FUNCTION_BLOCK AX_ATM_FB_TON (* standard timer function block (on-delay timing) with AX/ATM Adapter, PT and ET as adapters *)
  (* Standard: 61131-3; Classification: standard timer function block; Description: Copyright (c) 2026 HR Agrartechnik GmbH This program and the accompanying materials are made available under the terms of the Eclipse Public License 2.0 which is available at https://www.eclipse.org/legal/epl-2.0/ SPDX-License-Identifier: EPL-2.0 Wie AX_FB_TON, aber PT (Socket) und ET (Plug) sind ATM-Adapter statt einfacher Datenvariablen, damit sie ueber AR_SUBSCRIBE_1/AR_PUBLISH_1-artige Ketten mit REAL-Sekundenwerten verdrahtet werden koennen, ohne eigene Datenverbindungen fuer PT/ET zu brauchen. REQ bleibt ein einfaches Event - damit die Anwendung selbst einen E_CYCLE anschliessen kann, um ET periodisch zu aktualisieren, waehrend der Timer laeuft. ET feuert sein Adapterereignis nur bei tatsaechlicher Wertaenderung (E_D_FF_ANY), nicht bei jedem REQ. PT-Verhalten: PT.D1 liegt als reine Datenverbindung dauerhaft am internen FB_TON.PT an - der Adapter puffert/entprellt PT nicht. IN.E1, PT.E1 und das externe REQ sind gleichwertige Ausloeser fuer dieselbe FB_TON.REQ-Auswertung; FB_TON selbst unterscheidet nicht, welcher der drei es war. Eine Aenderung von PT ist also nicht am Start (steigende Flanke von IN) eingefroren, sondern wirkt bei der naechsten Auswertung sofort mit dem dann aktuellen ET zusammen - siehe Technische Besonderheiten in der Doku fuer die Grenzfaelle PT=0 und schnell aufeinanderfolgende PT-Aenderungen. Vor dem allerersten PT.E1 liegt an FB_TON.PT der TIME-Standardwert T#0s an, nicht ein projektspezifischer Default. *)
  (* Version 1.0, 2026-08-13, Franz Höpfinger, HR Agrartechnik GmbH, initial API and implementation *)
  PACKAGE adapter::iec61131::timers;
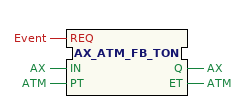
  EVENT_INPUT
    REQ; (* Normal Execution Request (non-triggering); gleichwertig zu IN.E1/PT.E1 (alle drei loesen dieselbe interne Neuauswertung aus). Anwendung haengt hier periodisch einen E_CYCLE an, damit ET auch ohne IN-/PT-Aenderung aktualisiert wird *)
  END_EVENT
  SOCKETS
    IN : adapter::types::unidirectional::AX; (* Input *)
    PT : adapter::types::unidirectional::ATM; (* Process time; live/nicht gelatched - PT.E1 loest wie IN.E1/REQ sofort eine Neuauswertung mit dem neuen PT-Wert aus, keine Entprellung. PT=0 laesst Q bei der naechsten Auswertung sofort TRUE werden *)
  END_SOCKETS
  PLUGS
    Q : adapter::types::unidirectional::AX; (* Output *)
    ET : adapter::types::unidirectional::ATM; (* Elapsed time, Event nur bei Wertaenderung *)
  END_PLUGS
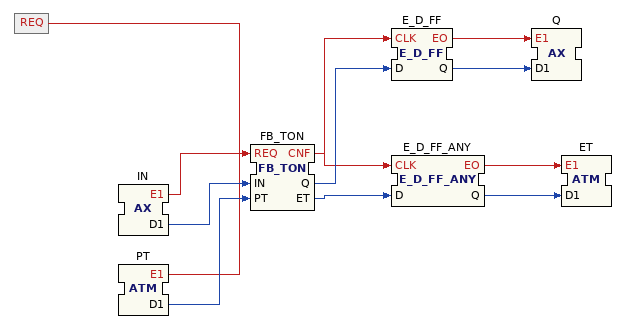
  FBS
    FB_TON : iec61131::timers::FB_TON;
    E_D_FF : iec61499::events::E_D_FF;
    E_D_FF_ANY : iec61499::events::E_D_FF_ANY;
  END_FBS
  EVENT_CONNECTIONS
    IN.E1 TO FB_TON.REQ;
    REQ TO FB_TON.REQ;
    FB_TON.CNF TO E_D_FF.CLK;
    E_D_FF.EO TO Q.E1;
    FB_TON.CNF TO E_D_FF_ANY.CLK;
    E_D_FF_ANY.EO TO ET.E1;
    PT.E1 TO FB_TON.REQ;
  END_CONNECTIONS
  DATA_CONNECTIONS
    IN.D1 TO FB_TON.IN;
    PT.D1 TO FB_TON.PT;
    FB_TON.Q TO E_D_FF.D;
    E_D_FF.Q TO Q.D1;
    FB_TON.ET TO E_D_FF_ANY.D;
    E_D_FF_ANY.Q TO ET.D1;
  END_CONNECTIONS
END_FUNCTION_BLOCK
